// TIA Portal V18 export
DATA_BLOCK "Utility_selection_DB"   // DB6
VERSION : 0.1
// stored: AutoNumber true, DBAccessibleFromOPCUA true, DBAccessibleFromWebserver true, InstanceOfName Utility_selection, InstanceOfType FB
"Utility_selection"
   // VAR_INPUT
   //    utl_type : Int;
   //    chbs_ofb : Bool;
   //    chbs_cfb : Bool;
   //    chws_ofb : Bool;
   //    chws_cfb : Bool;
   //    cws_ofb : Bool;
   //    cws_cfb : Bool;
   //    hws_ofb : Bool;
   //    hws_cfb : Bool;
   //    as_ofb : Bool;
   //    as_cfb : Bool;
   //    byp_ofb : Bool;
   //    byp_cfb : Bool;
   //    chbr_ofb : Bool;
   //    chbr_cfb : Bool;
   //    chwr_ofb : Bool;
   //    chwr_cfb : Bool;
   //    hwr_ofb : Bool;
   //    hwr_cfb : Bool;
   //    cwr_ofb : Bool;
   //    cwr_cfb : Bool;
   //    cond_ofb : Bool;
   //    cond_cfb : Bool;
   //    dr_ofb : Bool;
   //    dr_cfb : Bool;
   //    av_ofb : Bool;
   //    av_cfb : Bool;
   //    scv_ofb : Bool;
   //    times : Array[0..2] of DInt;
   // END_VAR
   // VAR_OUTPUT
   //    chbs_cmd : Bool;
   //    chws_cmd : Bool;
   //    cws_cmd : Bool;
   //    hws_cmd : Bool;
   //    as_cmd : Bool;
   //    byp_cmd : Bool;
   //    chbr_cmd : Bool;
   //    chwr_cmd : Bool;
   //    cwr_cmd : Bool;
   //    hwr_cmd : Bool;
   //    cond_cmd : Bool;
   //    dr_cmd : Bool;
   //    av_cmd : Bool;
   //    scv_cmd : Bool;
   //    flush_time : DInt;
   //    vent_time : DInt;
   //    drine_time : DInt;
   //    CMNR_cmd : Bool;
   // END_VAR
   // VAR_IN_OUT
   //    control { ExternalVisible := 'False'} : Word;
   //    utl_bit : Bool;
   // END_VAR
   // VAR
   //    selection : Int;
   //    br_sel : Bool;
   //    chw_sel : Bool;
   //    cw_sel : Bool;
   //    hw_sel : Bool;
   //    flush_sel : Bool;
   //    st_sel : Bool;
   //    prev_util : Int;
   //    vent_start : Bool;
   //    start_temp : Bool;
   //    start : Bool;
   //    flush_tm_comp : Bool;
   //    am : Bool;
   //    pause : Bool;
   //    chbr_cmd1 : Bool;
   //    chbr_cmd2 : Bool;
   //    agr_fail : Bool;
   //    hold : Bool;
   //    hold_t : Bool;
   //    status : Word;
   //    steam_flush : Bool;
   //    SUV_flush : Bool;
   //    Pres_low : Bool;
   //    uti_cv : Bool;
   //    hw_autoflush : Bool;
   //    emstop : Bool;
   //    temp : Bool;
   //    en_flush : Bool;
   //    dr_start : Bool;
   //    hwr_cmd1 : Bool;
   //    hwr_cmd2 : Bool;
   //    chwr_cmd1 : Bool;
   //    chwr_cmd2 : Bool;
   //    cond_cmd1 : Bool;
   //    cwr_cmd1 : Bool;
   //    cwr_cmd2 : Bool;
   //    br_flush : Bool;
   //    chw_flush : Bool;
   //    cw_flush : Bool;
   //    hw_flush : Bool;
   //    st_flush : Bool;
   //    byp_cmd2 : Bool;
   //    Flush_Dint : DInt;
   //    Flush_Ptime : Time;
   //    Flush_Etime : Time;
   //    Flush_TTime : DInt;
   //    Vent_Etime : Time;
   //    Vent_TTime : DInt;
   //    Vent_Ptime : Time;
   //    Vent_Dint : DInt;
   //    Cond_Dint : DInt;
   //    Cond_Ptime : Time;
   //    Cond_Etime : Time;
   //    Cond_TTime : DInt;
   //    reserved : Bool;
   //    Vent_tm_comp : Bool;
   //    Cond_tm_comp : Bool;
   //    US_TOF3 { S7_SetPoint := 'True'} : TOF_TIME;
   //    US_TON2 { S7_SetPoint := 'True'} : TON_TIME;
   //    US_TON3 { S7_SetPoint := 'True'} : TON_TIME;
   //    US_TON4 { S7_SetPoint := 'True'} : TON_TIME;
   //    US_TON5 { S7_SetPoint := 'True'} : TON_TIME;
   //    US_TP2 { S7_SetPoint := 'True'} : TP_TIME;
   //    US_TP3 { S7_SetPoint := 'True'} : TP_TIME;
   //    US_TP4 { S7_SetPoint := 'True'} : TP_TIME;
   //    US_TOF1 { S7_SetPoint := 'True'} : TOF_TIME;
   //    UP_TP6 { S7_SetPoint := 'True'} : TP_TIME;
   //    US_TP8 { S7_SetPoint := 'True'} : TP_TIME;
   //    US_TP7 { S7_SetPoint := 'True'} : TP_TIME;
   //    US_TP9 { S7_SetPoint := 'True'} : TP_TIME;
   //    UP_TP1 { S7_SetPoint := 'True'} : TP_TIME;
   //    US_TP10 { S7_SetPoint := 'True'} : TP_TIME;
   //    US_TOF2 { S7_SetPoint := 'True'} : TOF_TIME;
   //    US_TOF4 { S7_SetPoint := 'True'} : TOF_TIME;
   //    US_TOF6 { S7_SetPoint := 'True'} : TOF_TIME;
   //    US_TP11 { S7_SetPoint := 'True'} : TP_TIME;
   //    US_TP12 { S7_SetPoint := 'True'} : TP_TIME;
   //    US_TON6 { S7_SetPoint := 'True'} : TON_TIME;
   //    US_TP5 { S7_SetPoint := 'True'} : TP_TIME;
   //    US_TON7 { S7_SetPoint := 'True'} : TON_TIME;
   //    US_TP13 { S7_SetPoint := 'True'} : TP_TIME;
   //    US_TP14 { S7_SetPoint := 'True'} : TP_TIME;
   //    US_TON8 { S7_SetPoint := 'True'} : TON_TIME;
   //    US_TP15 { S7_SetPoint := 'True'} : TP_TIME;
   //    US_TP20 { S7_SetPoint := 'True'} : TP_TIME;
   //    US_TON10 { S7_SetPoint := 'True'} : TON_TIME;
   //    US_TP16 { S7_SetPoint := 'True'} : TP_TIME;
   //    US_TON9 { S7_SetPoint := 'True'} : TON_TIME;
   //    US_TP17 { S7_SetPoint := 'True'} : TP_TIME;
   //    US_TP21 { S7_SetPoint := 'True'} : TP_TIME;
   //    S_TON11 { S7_SetPoint := 'True'} : TON_TIME;
   //    US_TP18 { S7_SetPoint := 'True'} : TP_TIME;
   //    US_TP19 { S7_SetPoint := 'True'} : TP_TIME;
   // END_VAR
BEGIN
END_DATA_BLOCK
